(* Logix 5000 project; controller PLCbox vendor 1 type 14 code 149 rev 30.11; software revision 30.01; part 2 of 3 *)
(* tags used below, declared in another part *)
   ClearString : String20;
   FinalCode : String20;
   MyBarcode : STRING;
   OUT_Loc1_F : BOOL[32];
   OUT_Loc1_Index : DINT;
   OUT_S1 : UDT_Output[16];
   STR : STRING;
   test : DINT;
   test2 : DINT[2];
   HMI_Int_BOOL : BOOL[64];
   IN_Loc1 : BOOL[32];
   Light1_Complete_ONS : BOOL;
   Light1_Green : BOOL;
   Light1_Green_T : TIMER;
   Light1_Red : BOOL;
   Light1_Reset : BOOL;
   Light1_Yellow : BOOL;
   Light1_Yellow_T : TIMER;
   Light2_Complete_ONS : BOOL;
   Light2_Green : BOOL;
   Light2_Green_T : TIMER;
   Light2_Red : BOOL;
   Light2_Reset : BOOL;
   Light2_Yellow : BOOL;
   Light2_Yellow_T : TIMER;
   OUT_Loc1 : BOOL[32];
   PID_Analog_In : REAL[20];
   PLCTime : UDT_Time;
   Remote_Start_PB1 : ALIAS FOR PointIO_Rack1:1:I.0;
   Remote_Start_PB7 : ALIAS FOR PointIO_Rack1:1:I.0;
   Remote_STOP_PB1 : ALIAS FOR PointIO_Rack1:1:I.1;
   SsytemStopped : BOOL;
   StopBeacon : ALIAS FOR PointIO_Rack1:3:O.1;
(* MainProgram, continued *)

ROUTINE _03b_OutputLoop   (* ladder *)
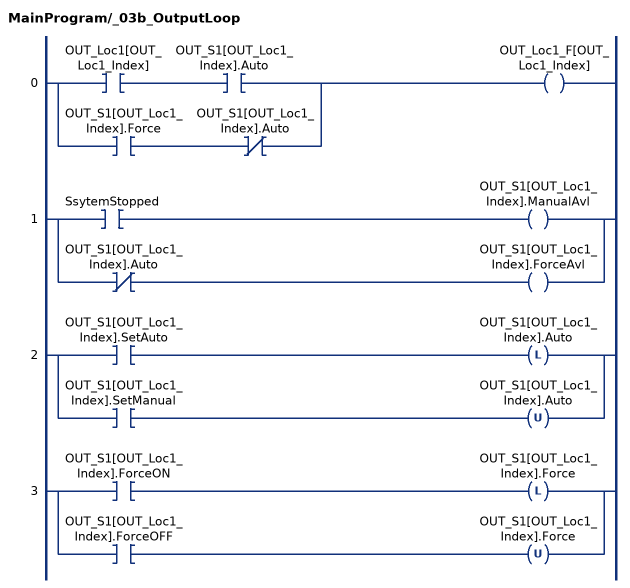
   0: [XIC(OUT_Loc1[OUT_Loc1_Index]) XIC(OUT_S1[OUT_Loc1_Index].Auto) ,XIC(OUT_S1[OUT_Loc1_Index].Force) XIO(OUT_S1[OUT_Loc1_Index].Auto) ]OTE(OUT_Loc1_F[OUT_Loc1_Index]);
   1: [XIC(SsytemStopped) OTE(OUT_S1[OUT_Loc1_Index].ManualAvl) ,XIO(OUT_S1[OUT_Loc1_Index].Auto) OTE(OUT_S1[OUT_Loc1_Index].ForceAvl) ];
   2: [XIC(OUT_S1[OUT_Loc1_Index].SetAuto) OTL(OUT_S1[OUT_Loc1_Index].Auto) ,XIC(OUT_S1[OUT_Loc1_Index].SetManual) OTU(OUT_S1[OUT_Loc1_Index].Auto) ];
   3: [XIC(OUT_S1[OUT_Loc1_Index].ForceON) OTL(OUT_S1[OUT_Loc1_Index].Force) ,XIC(OUT_S1[OUT_Loc1_Index].ForceOFF) OTU(OUT_S1[OUT_Loc1_Index].Force) ];
END_ROUTINE

ROUTINE _04_Cognex   (* ladder *)
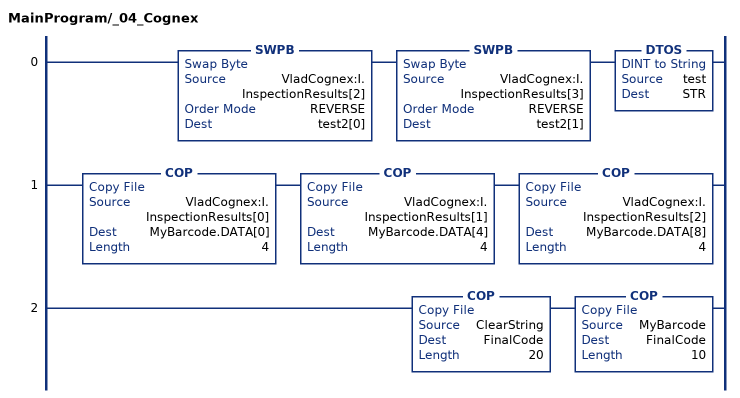
   0: SWPB(VladCognex:I.InspectionResults[2],REVERSE,test2[0])SWPB(VladCognex:I.InspectionResults[3],REVERSE,test2[1])DTOS(test,STR);
   1: COP(VladCognex:I.InspectionResults[0],MyBarcode.DATA[0],4)COP(VladCognex:I.InspectionResults[1],MyBarcode.DATA[4],4)COP(VladCognex:I.InspectionResults[2],MyBarcode.DATA[8],4);
   2: COP(ClearString,FinalCode,20)COP(MyBarcode,FinalCode,10);
END_ROUTINE

ROUTINE _05_General   (* ladder *)
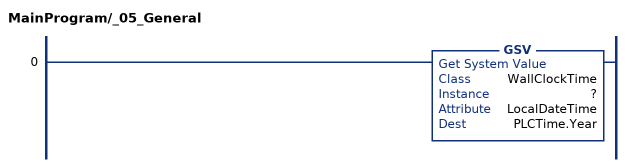
   0: GSV(WallClockTime,?,LocalDateTime,PLCTime.Year);
END_ROUTINE

ROUTINE _06_Ext_Inputs   (* ladder *)
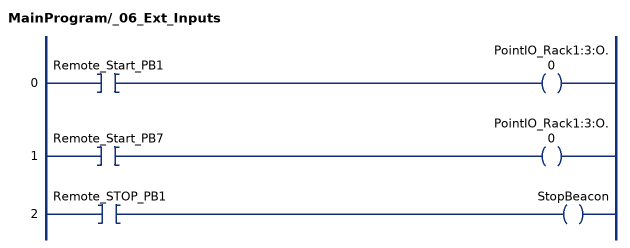
   0 (stored rung type 13): XIC(Remote_Start_PB1)OTE(PointIO_Rack1:3:O.0);
   1 (stored rung type 13): XIC(Remote_Start_PB7)OTE(PointIO_Rack1:3:O.0);
   2 (stored rung type 13): XIC(Remote_STOP_PB1)OTE(StopBeacon);
END_ROUTINE
END_PROGRAM

PROGRAM MainProgram2   (* main routine _01_Main *)
VAR
   PID_1001 : PID_ENHANCED := (PVEUMax := 100.0, SPOper := 50.0, SPHLimit := 100.0, RatioProg := 1.0, RatioOper := 1.0, RatioHLimit := 1.0, RatioLLimit := 1.0, CVOper := 100.0, CVEUMax := 100.0, CVHLimit := 100.0, DependIndepend := 1, PGain := 0.1, IGain := 0.001, DGain := 0.001, PVEDerivative := 1, ProgOperReq := 1, RTSTime := 1, CVEU := 100.0, CV := 100.0, CVHAlarm := 1, SP := 50.0, SPPercent := 50.0, E := 50.0, EPercent := 50.0, InitPrimary := 1, WindupHOut := 1, Ratio := 1.0, Auto := 1, DeltaT := 0.1);
   PID_Par_1001 : UDT_PID := (P := 0.1, I := 0.001, D := 0.001, CV := 100.0, SP := 50.0, Auto := 1, Name := 'PID 1001 - Testing CLICK PLC Input');
   SCL_01 : SCALE := (InRawMax := 5000.0, InEUMax := 100.0);
END_VAR

ROUTINE _01_Main   (* ladder *)
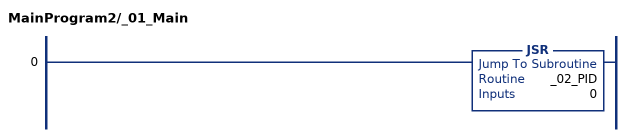
   0: JSR(_02_PID,0);
END_ROUTINE

ROUTINE _02_PID   (* function block diagram *)
   SHEET 1
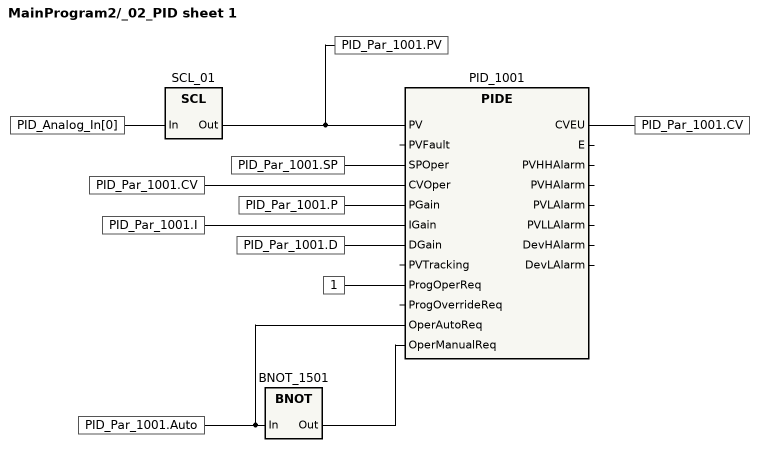
   SCL_01 : SCL(In := PID_Analog_In[0]);
   BNOT_1501 : BNOT(In := PID_Par_1001.Auto);
   PID_Par_1001.PV := SCL_01.Out;
   PID_1001 : PIDE(PV := SCL_01.Out, SPOper := PID_Par_1001.SP, CVOper := PID_Par_1001.CV, PGain := PID_Par_1001.P, IGain := PID_Par_1001.I, DGain := PID_Par_1001.D, ProgOperReq := 1, OperAutoReq := PID_Par_1001.Auto, OperManualReq := BNOT_1501.Out);   // unwired pins: PVFault PVTracking ProgOverrideReq E PVHHAlarm PVHAlarm PVLAlarm PVLLAlarm DevHAlarm DevLAlarm
   PID_Par_1001.CV := PID_1001.CVEU;
END_ROUTINE
END_PROGRAM

PROGRAM Mathematical   (* main routine _01_Main *)
VAR
   System_DINT : DINT[100] := ([0] := 12, [1] := 32, [2] := 54, [3] := 4, [4] := 31, [5] := 38, [6] := 100, [7] := 50, [8] := 200, [9] := 116);
   System_REAL : REAL[100] := ([0] := 23.0, [1] := 42.0, [2] := 0.48835304, [5] := 1.0);
END_VAR

ROUTINE _01_Main   (* ladder *)
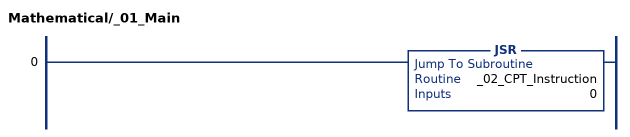
   0: JSR(_02_CPT_Instruction,0);
END_ROUTINE

ROUTINE _02_CPT_Instruction   (* ladder *)
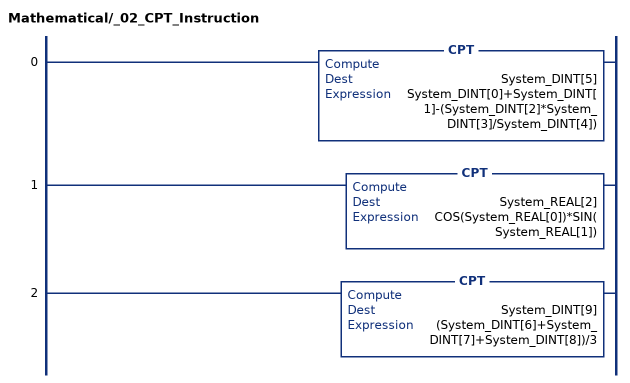
   0: CPT(System_DINT[5],System_DINT[0]+System_DINT[1]-(System_DINT[2]*System_DINT[3]/System_DINT[4]));
   1: CPT(System_REAL[2],COS(System_REAL[0])*SIN(System_REAL[1]));
   2: CPT(System_DINT[9],(System_DINT[6]+System_DINT[7]+System_DINT[8])/3);
END_ROUTINE
END_PROGRAM

PROGRAM PowerFlex525Mastery   (* main routine _01_Main *)
VAR
   Drive_Status : DINT := 2;
   Motor_Dev : REAL := 300.0;
   Motor_Fault_Timer : TIMER := (PRE := 20000);
   Motor_Faulted : BOOL := 1;
   Motor_Run : BOOL;
   Motor_SpdLim_High : REAL := 6300.0;
   Motor_SpdLim_Low : REAL := 5700.0;
   Motor_Target_Speed_Fault : BOOL;
   Reset_PB : BOOL;
   Start_PB : BOOL;
   Stop_PB : BOOL;
END_VAR

ROUTINE _01_Main   (* ladder *)
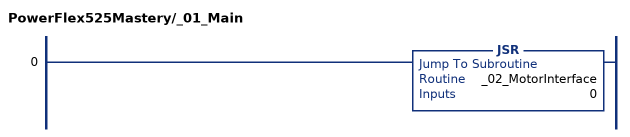
   0: JSR(_02_MotorInterface,0);
END_ROUTINE

ROUTINE _02_MotorInterface   (* ladder *)
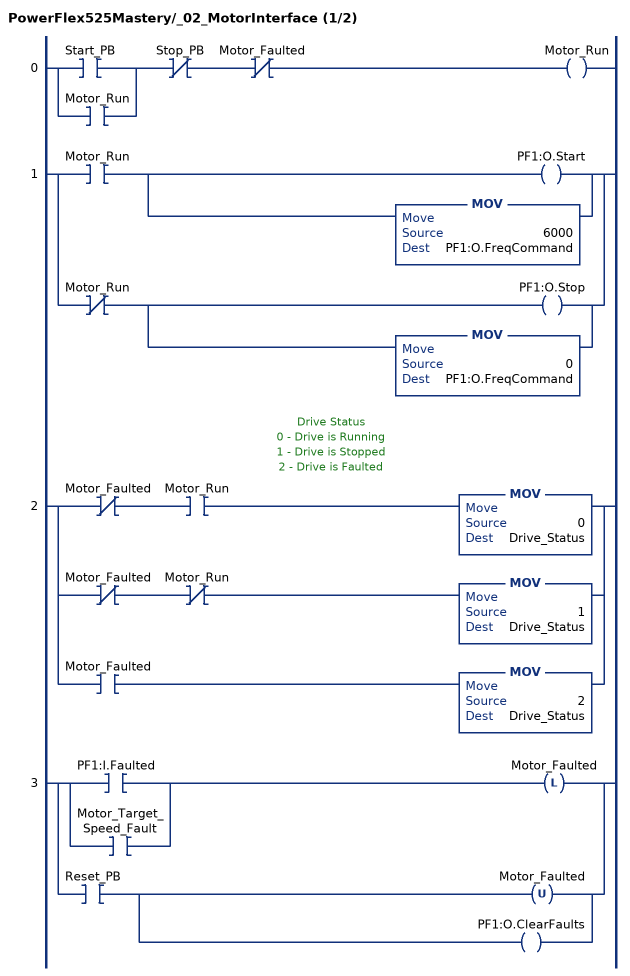
   0: [XIC(Start_PB) ,XIC(Motor_Run) ]XIO(Stop_PB)XIO(Motor_Faulted)OTE(Motor_Run);
   1: [XIC(Motor_Run) [OTE(PF1:O.Start) ,MOV(6000,PF1:O.FreqCommand) ] ,XIO(Motor_Run) [OTE(PF1:O.Stop) ,MOV(0,PF1:O.FreqCommand) ] ];
   // Drive Status
   // 0 - Drive is Running
   // 1 - Drive is Stopped
   // 2 - Drive is Faulted
   2: [XIO(Motor_Faulted) XIC(Motor_Run) MOV(0,Drive_Status) ,XIO(Motor_Faulted) XIO(Motor_Run) MOV(1,Drive_Status) ,XIC(Motor_Faulted) MOV(2,Drive_Status) ];
   3: [[XIC(PF1:I.Faulted) ,XIC(Motor_Target_Speed_Fault) ] OTL(Motor_Faulted) ,XIC(Reset_PB) [OTU(Motor_Faulted) ,OTE(PF1:O.ClearFaults) ] ];
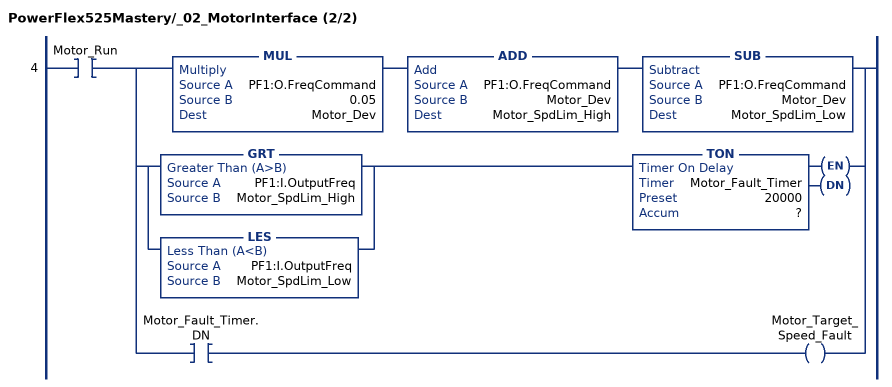
   4: XIC(Motor_Run)[MUL(PF1:O.FreqCommand,0.05,Motor_Dev) ADD(PF1:O.FreqCommand,Motor_Dev,Motor_SpdLim_High) SUB(PF1:O.FreqCommand,Motor_Dev,Motor_SpdLim_Low) ,[GRT(PF1:I.OutputFreq,Motor_SpdLim_High) ,LES(PF1:I.OutputFreq,Motor_SpdLim_Low) ] TON(Motor_Fault_Timer,?,?) ,XIC(Motor_Fault_Timer.DN) OTE(Motor_Target_Speed_Fault) ];
END_ROUTINE
END_PROGRAM

PROGRAM ST_Practice   (* main routine _01_Main *)
VAR
   MotorRUN : DINT;
   MotorRUN2 : BOOL := 1;
   MTR1 : BOOL[64];
        [0]   // Motor - Start PB
        [1]   // Motor - Stop PB
        [2]   // Motor - Running
   StartPB : BOOL;
   StopPB : DINT;
   StopPB2 : BOOL;
END_VAR

ROUTINE _01_Main   (* ladder *)
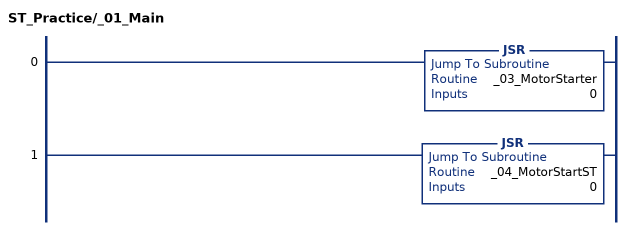
   0: JSR(_03_MotorStarter,0);
   1: JSR(_04_MotorStartST,0);
END_ROUTINE

ROUTINE _02_InputDef   (* structured text *)
   IN_Loc1[0] := Local:1:I.Data.0; //Start PB
   IN_Loc1[1] := Local:1:I.Data.1; //Stop PB
   IN_Loc1[2] := Local:1:I.Data.2; //Reset from HMI
   IN_Loc1[3] := Local:1:I.Data.3; //
   IN_Loc1[4] := Local:1:I.Data.4; //
   IN_Loc1[5] := Local:1:I.Data.5; //
   IN_Loc1[6] := Local:1:I.Data.6; //
   IN_Loc1[7] := Local:1:I.Data.7; //
   IN_Loc1[8] := Local:1:I.Data.8; //
   IN_Loc1[9] := Local:1:I.Data.9; //
   IN_Loc1[10] := Local:1:I.Data.10; //
   IN_Loc1[11] := Local:1:I.Data.11; //
   IN_Loc1[12] := Local:1:I.Data.12; //
   IN_Loc1[13] := Local:1:I.Data.13; //
   IN_Loc1[14] := Local:1:I.Data.14; //
   IN_Loc1[15] := Local:1:I.Data.15; //
END_ROUTINE

ROUTINE _03_MotorStarter   (* ladder *)
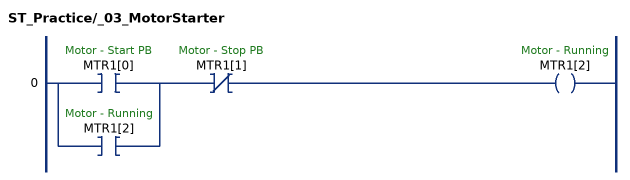
   0: [XIC(MTR1[0]) ,XIC(MTR1[2]) ]XIO(MTR1[1])OTE(MTR1[2]);
END_ROUTINE

ROUTINE _04_MotorStartST   (* structured text *)
   // MTR1[3] - StartPB
   // MTR1[4] - StopPB
   // MTR1[5] - Motor Running
   //MTR1[5] := (MTR1[3] OR MTR1[5]) AND NOT(MTR1[4]);
   IF (MTR1[3] OR MTR1[5]) AND NOT(MTR1[4]) THEN
   MTR1[5] := 1;
   ELSE
   MTR1[5] := 0;
   END_IF;
END_ROUTINE
END_PROGRAM

PROGRAM StreetLightSystem   (* main routine _01_Main *)
VAR
   HMI_Int_DINT : DINT[100] := ([0] := 10000, [1] := 3000, [2] := 10000, [3] := 3000);
END_VAR

ROUTINE _01_Main   (* ladder *)
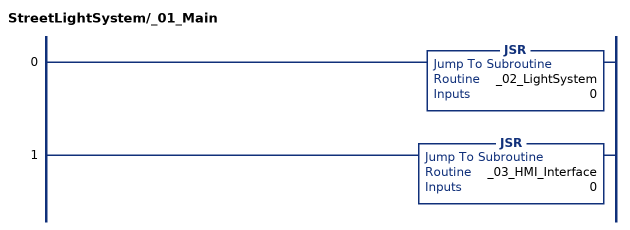
   0: JSR(_02_LightSystem,0);
   1: JSR(_03_HMI_Interface,0);
END_ROUTINE

ROUTINE _02_LightSystem   (* ladder *)
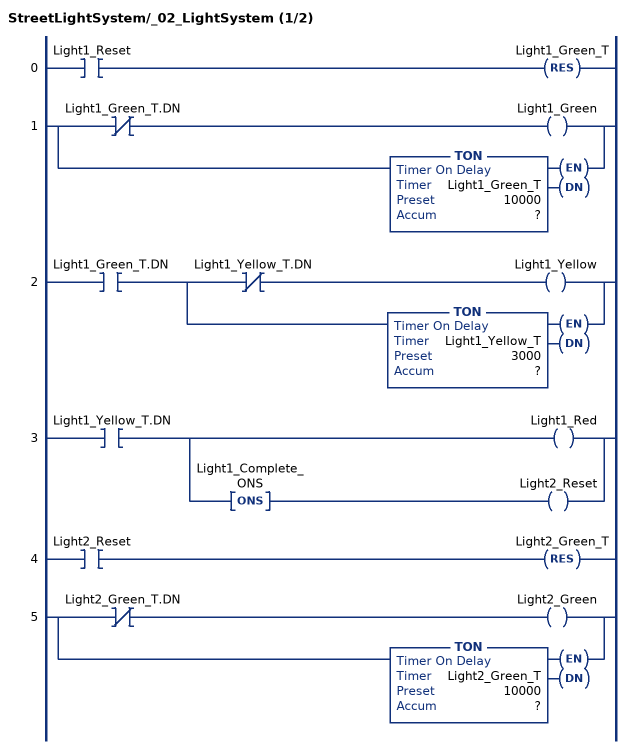
   0: XIC(Light1_Reset)RES(Light1_Green_T);
   1: [XIO(Light1_Green_T.DN) OTE(Light1_Green) ,TON(Light1_Green_T,?,?) ];
   2: XIC(Light1_Green_T.DN)[XIO(Light1_Yellow_T.DN) OTE(Light1_Yellow) ,TON(Light1_Yellow_T,?,?) ];
   3: XIC(Light1_Yellow_T.DN)[OTE(Light1_Red) ,ONS(Light1_Complete_ONS) OTE(Light2_Reset) ];
   4: XIC(Light2_Reset)RES(Light2_Green_T);
   5: [XIO(Light2_Green_T.DN) OTE(Light2_Green) ,TON(Light2_Green_T,?,?) ];
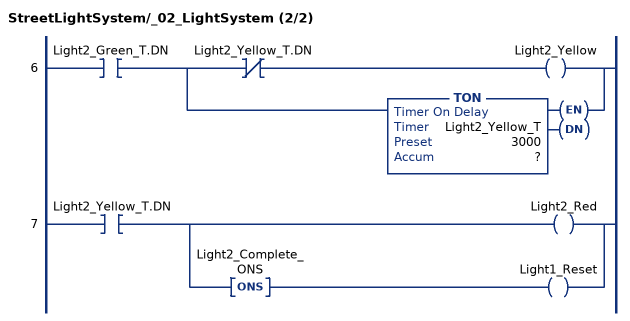
   6: XIC(Light2_Green_T.DN)[XIO(Light2_Yellow_T.DN) OTE(Light2_Yellow) ,TON(Light2_Yellow_T,?,?) ];
   7: XIC(Light2_Yellow_T.DN)[OTE(Light2_Red) ,ONS(Light2_Complete_ONS) OTE(Light1_Reset) ];
END_ROUTINE

ROUTINE _03_HMI_Interface   (* ladder *)
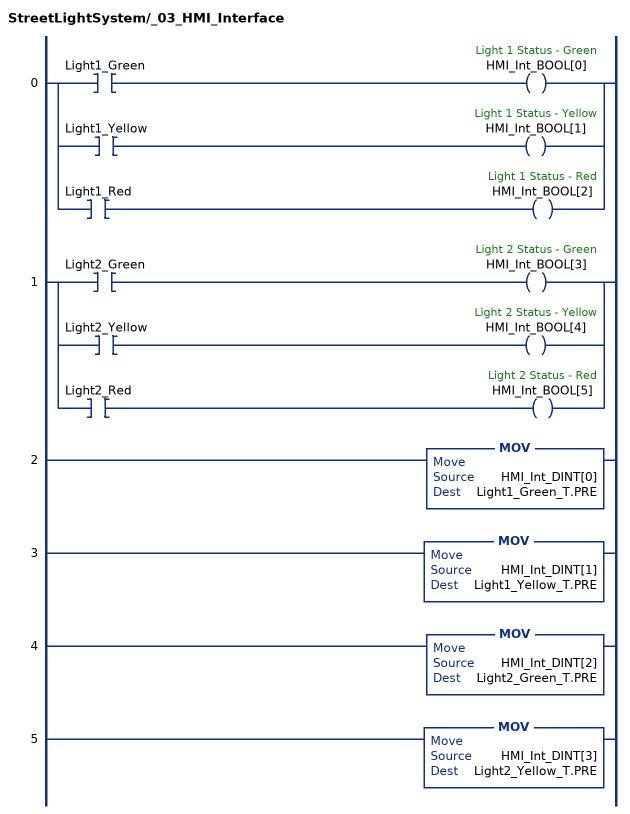
   0: [XIC(Light1_Green) OTE(HMI_Int_BOOL[0]) ,XIC(Light1_Yellow) OTE(HMI_Int_BOOL[1]) ,XIC(Light1_Red) OTE(HMI_Int_BOOL[2]) ];
   1: [XIC(Light2_Green) OTE(HMI_Int_BOOL[3]) ,XIC(Light2_Yellow) OTE(HMI_Int_BOOL[4]) ,XIC(Light2_Red) OTE(HMI_Int_BOOL[5]) ];
   2: MOV(HMI_Int_DINT[0],Light1_Green_T.PRE);
   3: MOV(HMI_Int_DINT[1],Light1_Yellow_T.PRE);
   4: MOV(HMI_Int_DINT[2],Light2_Green_T.PRE);
   5: MOV(HMI_Int_DINT[3],Light2_Yellow_T.PRE);
END_ROUTINE
END_PROGRAM

PROGRAM TankFillingChallenge   (* main routine _01_Main *)
VAR
   DischargeStatus : DINT := 1;
   FillingStatus : DINT := 1;
   T_Vlad : BOOL[128];
   TankActualLevel : REAL := 42.792046;
   TankDischargeRate : REAL := 0.5;
   TankEmptyThreshold : REAL := 5.0;
   TankFill : BOOL[128];
        [0]   // START Filling Station
        [1]   // STOP Filling Station
        [2]   // Filling Station RUNNING
        [3]   // START Discharge Station
        [4]   // STOP Discharge Station
        [5]   // Discharge Station RUNNING
        [6]   // TANK FULL
        [7]   // TANK EMPTY
   TankFillRate : REAL := 0.3;
   TankFullThreshold : REAL := 100.0;
   TankOut : BOOL[32];
        [0]   // Filling Station VALVE OPEN
        [1]   // Discharge Station VALVE OPEN
   TankTimers : TIMER[10] := ([0].PRE := 20, [1].PRE := 20);
END_VAR

ROUTINE _01_Main   (* ladder *)
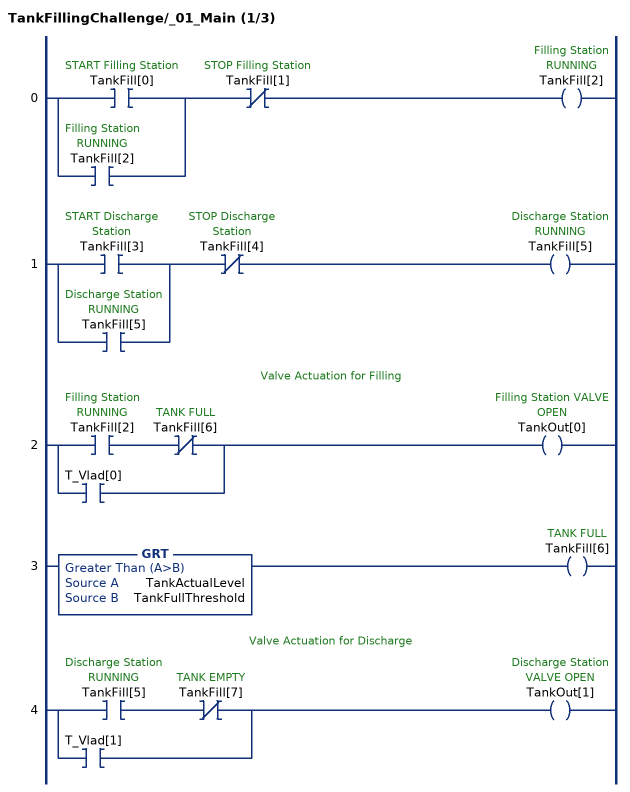
   0: [XIC(TankFill[0]) ,XIC(TankFill[2]) ]XIO(TankFill[1])OTE(TankFill[2]);
   1: [XIC(TankFill[3]) ,XIC(TankFill[5]) ]XIO(TankFill[4])OTE(TankFill[5]);
   // Valve Actuation for Filling
   2: [XIC(TankFill[2]) XIO(TankFill[6]) ,XIC(T_Vlad[0]) ]OTE(TankOut[0]);
   3: GRT(TankActualLevel,TankFullThreshold)OTE(TankFill[6]);
   // Valve Actuation for Discharge
   4: [XIC(TankFill[5]) XIO(TankFill[7]) ,XIC(T_Vlad[1]) ]OTE(TankOut[1]);
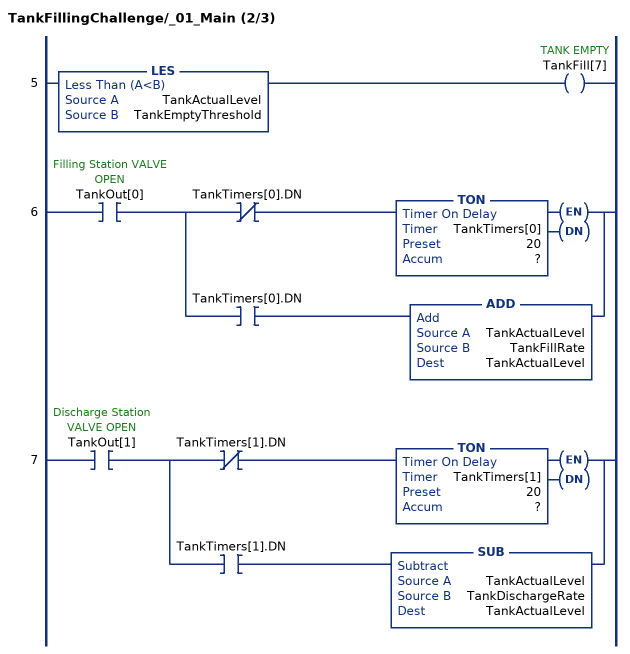
   5: LES(TankActualLevel,TankEmptyThreshold)OTE(TankFill[7]);
   6: XIC(TankOut[0])[XIO(TankTimers[0].DN) TON(TankTimers[0],?,?) ,XIC(TankTimers[0].DN) ADD(TankActualLevel,TankFillRate,TankActualLevel) ];
   7: XIC(TankOut[1])[XIO(TankTimers[1].DN) TON(TankTimers[1],?,?) ,XIC(TankTimers[1].DN) SUB(TankActualLevel,TankDischargeRate,TankActualLevel) ];
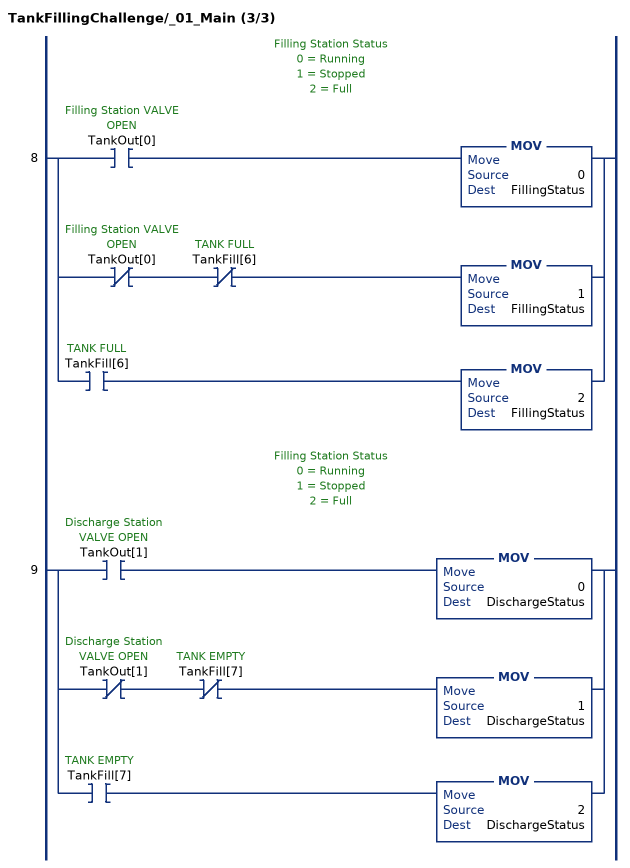
   // Filling Station Status
   // 0 = Running
   // 1 = Stopped
   // 2 = Full
   8: [XIC(TankOut[0]) MOV(0,FillingStatus) ,XIO(TankOut[0]) XIO(TankFill[6]) MOV(1,FillingStatus) ,XIC(TankFill[6]) MOV(2,FillingStatus) ];
   // Filling Station Status
   // 0 = Running
   // 1 = Stopped
   // 2 = Full
   9: [XIC(TankOut[1]) MOV(0,DischargeStatus) ,XIO(TankOut[1]) XIO(TankFill[7]) MOV(1,DischargeStatus) ,XIC(TankFill[7]) MOV(2,DischargeStatus) ];
END_ROUTINE
END_PROGRAM
